(* Schneider Machine Expert - Basic project simulation, file version 2.2.0.0 *)
(* ProjectInformations: Name=New project *)

HARDWARE
  Cpu 0: TM221ME16R/G
  EthernetConfiguration: NetworkName=M221, IpAllocationMode=FixedAddress, IpAddress=0.0.0.0, SubnetMask=0.0.0.0
  SerialLineConfiguration: Baud=Baud19200, Parity=ParityEven, DataBits=DataBits8, StopBits=StopBits1, PhysicalMedium=PhysicalMediumRs485, TransmissionMode=TransmissionModeModbusRtu, SlaveId=1, Addressing=SlaveAddressing
  MastTask: UsePeriodScanMode=false, PeriodScan=100
  FastTask: Period=255
  CpuBehavior: StartingMode=StartAsPreviousState, AutoSaveRamOnEeprom=true, WatchdogPeriod=250

SYMBOLS  (address, symbol, comment, settings)
  %M0       MIXING_TANK_INLET_VALVE_1
  %M1       MIXING_TANK_INLET_VALVE_2
  %M2       MIXING_TANK_OUTLET_VALVE
  %M3       STORAGE_TANK_INLET_VALVE
  %M4       AGITATOR_START
  %M5       PUMP_START
  %M6       PROCESS_START
  %M7       MIX_FINISHED
  %MW0      AGITATOR_TARGET_RPM
  %MW1      PUMP_TARGET_RPM
  %MW2      PRODUCT_1_VOLUME
  %MW3      PRODUCT_2_VOLUME
  %MW4      TARGET_VOLUME
  %MW5      MIXING_TIME
  %MW10     MIXING_TANK_LEVEL
  %MW11     DESTINATION_TANK_LEVEL
  %MW12     AGITATOR_REAL_RPM
  %MW13     PUMP_REAL_RPM
  %MD0      TEST_DECIMAL
  %TM1        [Preset=60, Base=OneSecond]

POU New POU
  (* SectionNumber=1 *)

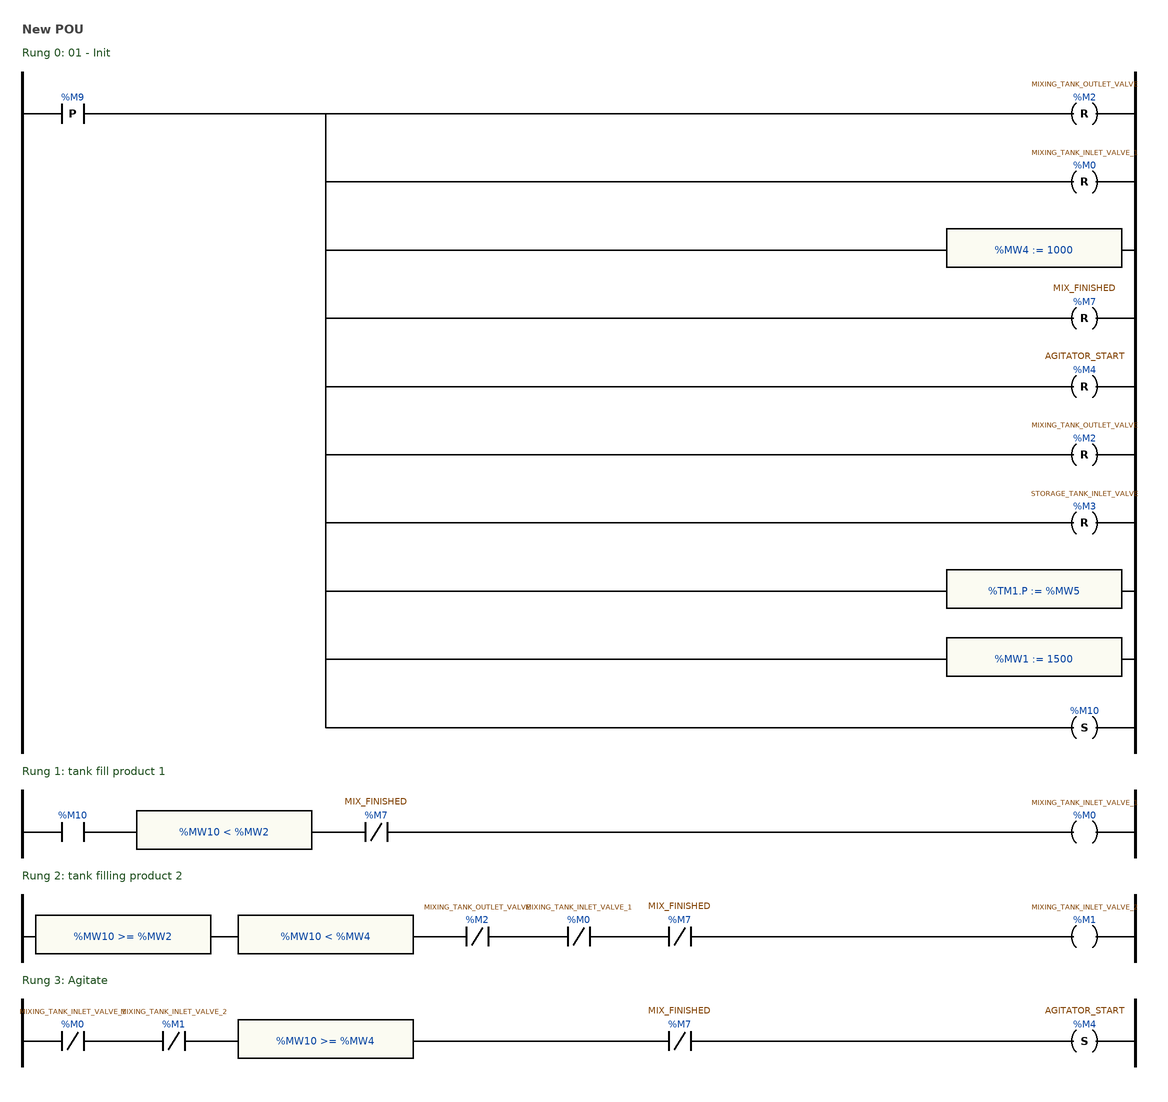

// Rung 0: 01 - Init
  LDR %M9
  R %M2                   (* MIXING_TANK_OUTLET_VALVE *)
  R %M0                   (* MIXING_TANK_INLET_VALVE_1 *)
  [ %MW4 := 1000 ]        (* TARGET_VOLUME *)
  R %M7                   (* MIX_FINISHED *)
  R %M4                   (* AGITATOR_START *)
  R %M2                   (* MIXING_TANK_OUTLET_VALVE *)
  R %M3                   (* STORAGE_TANK_INLET_VALVE *)
  [ %TM1.P := %MW5 ]      (* MIXING_TIME *)
  [ %MW1 := 1500 ]        (* PUMP_TARGET_RPM *)
  S %M10
  // as ST:
  //   IF RISING(%M9) THEN MIXING_TANK_OUTLET_VALVE := FALSE; END_IF;
  //   IF RISING(%M9) THEN MIXING_TANK_INLET_VALVE_1 := FALSE; END_IF;
  //   IF RISING(%M9) THEN TARGET_VOLUME := 1000; END_IF;
  //   IF RISING(%M9) THEN MIX_FINISHED := FALSE; END_IF;
  //   IF RISING(%M9) THEN AGITATOR_START := FALSE; END_IF;
  //   IF RISING(%M9) THEN MIXING_TANK_OUTLET_VALVE := FALSE; END_IF;
  //   IF RISING(%M9) THEN STORAGE_TANK_INLET_VALVE := FALSE; END_IF;
  //   IF RISING(%M9) THEN %TM1.P := MIXING_TIME; END_IF;
  //   IF RISING(%M9) THEN PUMP_TARGET_RPM := 1500; END_IF;
  //   IF RISING(%M9) THEN %M10 := TRUE; END_IF;

// Rung 1: tank fill product 1
  LD %M10
  AND [ %MW10 < %MW2 ]    (* MIXING_TANK_LEVEL, PRODUCT_1_VOLUME *)
  ANDN %M7                (* MIX_FINISHED *)
  ST %M0                  (* MIXING_TANK_INLET_VALVE_1 *)
  // as ST:
  //   MIXING_TANK_INLET_VALVE_1 := %M10 AND MIXING_TANK_LEVEL < PRODUCT_1_VOLUME AND NOT MIX_FINISHED;

// Rung 2: tank filling product 2
  LD [ %MW10 >= %MW2 ]    (* MIXING_TANK_LEVEL, PRODUCT_1_VOLUME *)
  AND [ %MW10 < %MW4 ]    (* MIXING_TANK_LEVEL, TARGET_VOLUME *)
  ANDN %M2                (* MIXING_TANK_OUTLET_VALVE *)
  ANDN %M0                (* MIXING_TANK_INLET_VALVE_1 *)
  ANDN %M7                (* MIX_FINISHED *)
  ST %M1                  (* MIXING_TANK_INLET_VALVE_2 *)
  // as ST:
  //   MIXING_TANK_INLET_VALVE_2 := MIXING_TANK_LEVEL >= PRODUCT_1_VOLUME AND MIXING_TANK_LEVEL < TARGET_VOLUME AND NOT MIXING_TANK_OUTLET_VALVE AND NOT MIXING_TANK_INLET_VALVE_1 AND NOT MIX_FINISHED;

// Rung 3: Agitate
  LDN %M0                 (* MIXING_TANK_INLET_VALVE_1 *)
  ANDN %M1                (* MIXING_TANK_INLET_VALVE_2 *)
  AND [ %MW10 >= %MW4 ]   (* MIXING_TANK_LEVEL, TARGET_VOLUME *)
  ANDN %M7                (* MIX_FINISHED *)
  S %M4                   (* AGITATOR_START *)
  // as ST:
  //   IF NOT MIXING_TANK_INLET_VALVE_1 AND NOT MIXING_TANK_INLET_VALVE_2 AND MIXING_TANK_LEVEL >= TARGET_VOLUME AND NOT MIX_FINISHED THEN AGITATOR_START := TRUE; END_IF;

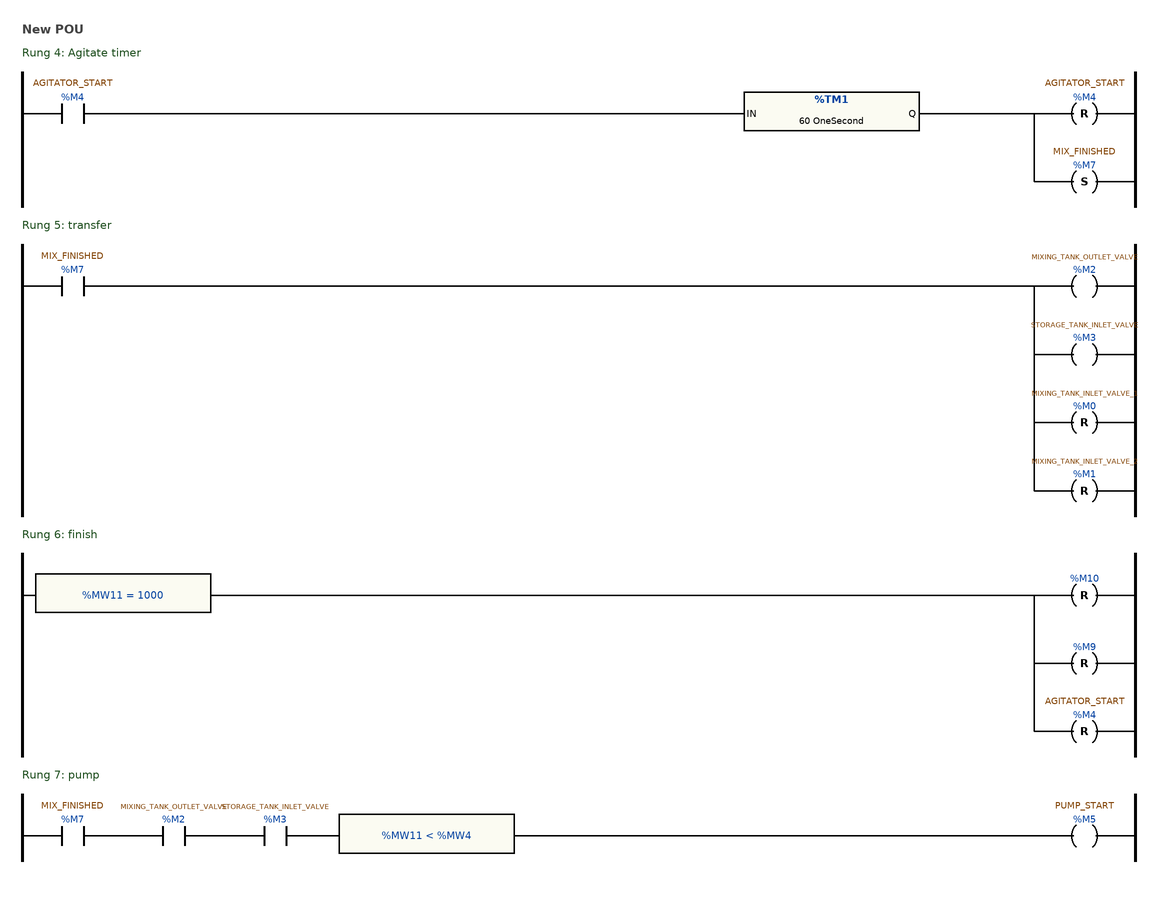

// Rung 4: Agitate timer
  BLK %TM1
  LD %M4                  (* AGITATOR_START *)
  IN
  OUT_BLK
  LD Q
  R %M4                   (* AGITATOR_START *)
  S %M7                   (* MIX_FINISHED *)
  END_BLK
  // as ST:
  //   %TM1(IN := AGITATOR_START);
  //   IF %TM1.Q THEN AGITATOR_START := FALSE; END_IF;
  //   IF %TM1.Q THEN MIX_FINISHED := TRUE; END_IF;

// Rung 5: transfer
  LD %M7                  (* MIX_FINISHED *)
  ST %M2                  (* MIXING_TANK_OUTLET_VALVE *)
  ST %M3                  (* STORAGE_TANK_INLET_VALVE *)
  R %M0                   (* MIXING_TANK_INLET_VALVE_1 *)
  R %M1                   (* MIXING_TANK_INLET_VALVE_2 *)
  // as ST:
  //   MIXING_TANK_OUTLET_VALVE := MIX_FINISHED;
  //   STORAGE_TANK_INLET_VALVE := MIX_FINISHED;
  //   IF MIX_FINISHED THEN MIXING_TANK_INLET_VALVE_1 := FALSE; END_IF;
  //   IF MIX_FINISHED THEN MIXING_TANK_INLET_VALVE_2 := FALSE; END_IF;

// Rung 6: finish
  LD [ %MW11 = 1000 ]     (* DESTINATION_TANK_LEVEL *)
  R %M10
  R %M9
  R %M4                   (* AGITATOR_START *)
  // as ST:
  //   IF DESTINATION_TANK_LEVEL = 1000 THEN %M10 := FALSE; END_IF;
  //   IF DESTINATION_TANK_LEVEL = 1000 THEN %M9 := FALSE; END_IF;
  //   IF DESTINATION_TANK_LEVEL = 1000 THEN AGITATOR_START := FALSE; END_IF;

// Rung 7: pump
  LD %M7                  (* MIX_FINISHED *)
  AND %M2                 (* MIXING_TANK_OUTLET_VALVE *)
  AND %M3                 (* STORAGE_TANK_INLET_VALVE *)
  AND [ %MW11 < %MW4 ]    (* DESTINATION_TANK_LEVEL, TARGET_VOLUME *)
  ST %M5                  (* PUMP_START *)
  // as ST:
  //   PUMP_START := MIX_FINISHED AND MIXING_TANK_OUTLET_VALVE AND STORAGE_TANK_INLET_VALVE AND DESTINATION_TANK_LEVEL < TARGET_VOLUME;
